(* IEC 61131-3 sources: AXOpen/src/components.festo.drives/ctrl/src/AxoCmmtAs/TypesStructuresAndEnums, 4 files *)

(* ---- AxoCmmtAs_Component_Status.st ---- *)
NAMESPACE AXOpen.Components.Festo.Drives
    {S7.extern=ReadWrite}
    {#ix-attr:[Container(Layout.Stack)]}
    // CLASS PUBLIC AxoCmmtAs EXTENDS AXOpen.Components.Abstractions.AxoComponent_Status
    //     VAR PUBLIC

    //     END_VAR
    // END_CLASS
    CLASS PUBLIC AxoCmmtAs_Component_Status EXTENDS AXOpen.Components.Drives.AxoDrive_Status
        VAR PUBLIC

        END_VAR
    END_CLASS
END_NAMESPACE

(* ---- AxoCmmtAsAxisData.st ---- *)
NAMESPACE AXOpen.Components.Festo.Drives
    {S7.extern=ReadWrite}
    CLASS AxoCmmtAsAxisData
        VAR PUBLIC
            // hwID                        :   WORD;
            // hwIdModuleAccessPoint       :   WORD;
            // hwIdTelegram111             :   WORD;
            // hwIdTelegram750             :   WORD;
            Cycle                       :   ULINT;
            OverrideVelocityFactor		:	LREAL := 1.0;	//LREAL value to be written
            OverrideAccelerationFactor	:	LREAL := 1.0;	//LREAL value to be written
            OverrideJerkFactor			:	LREAL := 1.0;	//LREAL value to be written
        END_VAR
    END_CLASS
END_NAMESPACE

(* ---- AxoCmmtAsAxisHWIDs.st ---- *)
NAMESPACE AXOpen.Components.Festo.Drives
   {S7.extern=ReadWrite}
	CLASS AxoCmmtAsAxisHWIDs
      VAR PUBLIC
         {#ix-set:AttributeName = "<#Hardware ID Device#>"}
         HW_Device            : UINT;
         {#ix-set:AttributeName = "<#Hardware ID 'DoServo' module#>"}
         HW_DoServo           : UINT;
         {#ix-set:AttributeName = "<#Hardware ID 'DoServo' submodule#>"}
         HW_DoServoSub           : UINT;
         {#ix-set:AttributeName = "<#Hardware ID 'ModuleAccessPoint' module#>"}
         HW_ModuleAccessPoint : UINT;
         {#ix-set:AttributeName = "<#Hardware ID 'EmptyModule_1' submodule#>"}
         HW_EmptyModule_1     : UINT;
         {#ix-set:AttributeName = "<#Hardware ID 'Telegram111' submodule#>"}
         HW_Telegram111       : UINT;
         {#ix-set:AttributeName = "<#Hardware ID 'EmptyModule_2' submodule#>"}
         HW_EmptyModule_2     : UINT;
         {#ix-set:AttributeName = "<#Hardware ID 'Telegram750' submodule#>"}
         HW_Telegram750       : UINT;
      END_VAR
   END_CLASS
END_NAMESPACE

(* ---- AxoCmmtAsAxisReference.st ---- *)
NAMESPACE AXOpen.Components.Festo.Drives
    {S7.extern=ReadWrite}
    {#ix-attr:[Container(Layout.Tabs)]}
    CLASS AxoCmmtAsAxisReference IMPLEMENTS AXOpen.Components.Abstractions.Drives.IAxoAxisReference
        VAR PUBLIC // Telegram 111
            {#ix-attr:[Container(Layout.Stack)]}
            {#ix-attr:[ComponentDetails("Telegram 111")]}
            {#ix-attr:[ReadOnly()]}
            {#ix-set:AttributeName = "<#Telegram111 Inputs#>"}
            Telegram111_In  :   AXOpen.Components.Festo.Drives.PROFIdriveTelegram_111_IN;
            {#ix-attr:[Container(Layout.Stack)]}
            {#ix-attr:[ComponentDetails("Telegram 111")]}
            // {#ix-attr:[ReadOnly()]}
            {#ix-set:AttributeName = "<#Telegram111 Outputs#>"}
            Telegram111_Out :   AXOpen.Components.Festo.Drives.PROFIdriveTelegram_111_OUT;
        END_VAR
        VAR PUBLIC // Telegram 750
            {#ix-attr:[Container(Layout.Stack)]}
            {#ix-attr:[ComponentDetails("Telegram 750")]}
            {#ix-attr:[ReadOnly()]}
            {#ix-set:AttributeName = "<#Telegram750 Inputs#>"}
            Telegram750_In  :   AXOpen.Components.Festo.Drives.PROFIdriveTelegram_750_IN;
            {#ix-attr:[Container(Layout.Stack)]}
            {#ix-attr:[ComponentDetails("Telegram 750")]}
            // {#ix-attr:[ReadOnly()]}
            {#ix-set:AttributeName = "<#Telegram750 Outputs#>"}
            Telegram750_Out :   AXOpen.Components.Festo.Drives.PROFIdriveTelegram_750_OUT;
        END_VAR
        VAR PUBLIC // HWIDs
            {#ix-attr:[Container(Layout.Stack)]}
            {#ix-attr:[ComponentDetails("HWids")]}
            {#ix-attr:[ReadOnly()]}
            HWIDs  :   AXOpen.Components.Festo.Drives.AxoCmmtAsAxisHWIDs;
        END_VAR
        VAR PUBLIC // Data
            {#ix-attr:[Container(Layout.Stack)]}
            {#ix-attr:[ComponentDetails("Data")]}
            {#ix-attr:[ReadOnly()]}
            Data            :   AXOpen.Components.Festo.Drives.AxoCmmtAsAxisData;
        END_VAR
        VAR PUBLIC
            Config          :   AXOpen.Components.Drives.AxoDrive_Config;
            Status          :   AXOpen.Components.Drives.AxoDrive_Status;
        END_VAR
    END_CLASS
END_NAMESPACE
